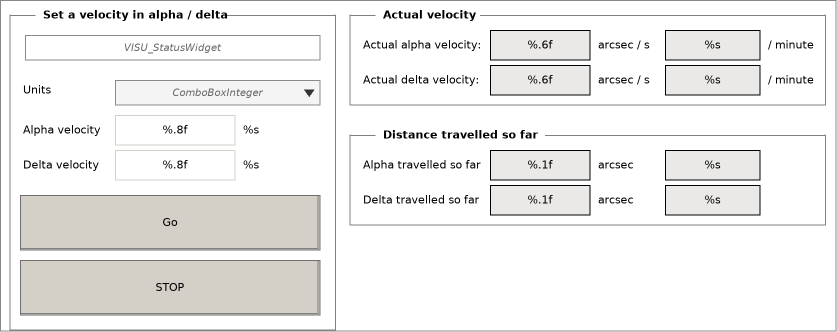
VISUALIZATION VISU_AxesManual_MoveVelocity  // 837x332
VAR_IN_OUT
	ref : Axes;
    widget : AxesManualMoveVelocityWidget;
END_VAR
    Polyline (225,15) (335,15) (335,330) (10,330) (10,15) (35,15)
    Polyline (480,15) (825,15) (825,105) (350,105) (350,15) (375,15)
    Label (380,5 100x20), "Actual velocity"
    Label (380,125 155x20), "Distance travelled so far"
    Polyline (545,135) (825,135) (825,225) (350,225) (350,135) (375,135)
    Textfield (115,115 120x30), "%.8f", text variable: widget.field_alphaVelocity
        OnMouseClick: write the text variable via VisuDialogs.Numpad
    Label (20,115 95x30), "Alpha velocity"
    Textfield (115,150 120x30), "%.8f", text variable: widget.field_deltaVelocity
        OnMouseClick: write the text variable via VisuDialogs.Numpad
    Label (20,150 95x30), "Delta velocity"
    Button (20,195 300x55), "Go", input disabled if: ref.processes.setAlphaDeltaVelocity.statuses.enabledStatus.disabled
        OnMouseClick: execute { widget.do_start := TRUE; }
    ComboBoxInteger (115,80 205x25), variable: widget.field_units, text list: 'AxesMoveVelocityUnitsTextList'
    Frame (25,35 295x25)
        shows VISU_StatusWidget(widget := widget.setAlphaDeltaVelocityStatus)
    Label (20,75 95x30), "Units"
    Rectangle (240,115 80x30), "%s", text variable: widget.label_units
    Label (360,30 145x30), "Actual alpha velocity:"
    Label (360,65 145x30), "Actual delta velocity:"
    Rectangle (490,30 100x30), "%.6f", text variable: ref.target.alphaVelocity.arcsecondsPerSecond.value
    Rectangle (490,65 100x30), "%.6f", text variable: ref.target.deltaVelocity.arcsecondsPerSecond.value
    Label (595,30 65x30), "arcsec / s"
    Rectangle (665,30 95x30), "%s", text variable: widget.alphaPerMinute.hmsString
    Rectangle (665,65 95x30), "%s", text variable: widget.deltaPerMinute.dmsString
    Label (765,30 70x30), "/ minute"
    Label (360,185 145x30), "Delta travelled so far"
    Label (360,150 145x30), "Alpha travelled so far"
    Rectangle (490,150 100x30), "%.1f", text variable: ref.target.alphaTravelled.arcseconds.value
    Rectangle (490,185 100x30), "%.1f", text variable: ref.target.deltaTravelled.arcseconds.value
    Label (595,150 75x30), "arcsec"
    Label (595,65 65x30), "arcsec / s"
    Label (765,65 70x30), "/ minute"
    Label (595,185 75x30), "arcsec"
    Rectangle (665,185 95x30), "%s", text variable: widget.deltaTravelledSoFar.dmsString
    Rectangle (665,150 95x30), "%s", text variable: widget.alphaTravelledSoFar.hmsString
    Button (20,260 300x55), "STOP", input disabled if: ref.processes.setAlphaDeltaVelocity.statuses.enabledStatus.disabled
        OnMouseClick: execute { widget.do_stop := TRUE; }
    Rectangle (240,150 80x30), "%s", text variable: widget.label_units
    Label (40,5 180x20), "Set a velocity in alpha / delta"
END_VISUALIZATION

(* stored: Version 1.1.0.1, ProductVersion 3.1.4019.2
   Visu VISU_AxesManual_MoveVelocity: Id {0452b5fe-ae1c-4ad5-8aef-b15436168b0b} *)
